{attribute 'GeneratedUsingTerminal: EP1518-0002-0016'}
{attribute addProperty BoxType "EP1518-0002-0016"}
{attribute addProperty Id "StatusAT %I*Status_D4FDECD45"}
{attribute addProperty CRC "525234923"}
{attribute addProperty Size "5"}
TYPE DIG_Inputs_Device_1F4E72EB EXTENDS InputBase_8311D824 :
STRUCT
	{attribute addProperty Name "Status"}
	Status AT %I* : Status_D4FDECD4;
END_STRUCT
END_TYPE

(* stored: Version 1.2.0.0, ProductVersion 3.1.4024.11
   DUT DIG_Inputs_Device_1F4E72EB: Id {6bc81971-e770-4ba5-b5c2-8359132e1ac7} *)
